{attribute addProperty BoxType "EK1100-0000-0018"}
{attribute addProperty Id "Beckhoff_ELXxxxxEK1122Beckhoff_ELXxxxxEK1122_CE175A58162A_0001_ELX1052_0000_0016ELX1052_F21EA95A506.25A_0002_ELX1054_0000_0016ELX1054_E012CCE111414.25A_0003_ELX1058_0000_0016ELX1058_D4A7C46F21026.25A_0004_ELX2002_0000_0016ELX2002_39EC201D334.125A_0005_ELX2008_0000_0016ELX2008_A854BE6D8110.125A_0006_ELX3152_0000_0016ELX3152_C6F348DD14618.25A_0007_ELX3152_0000_0017ELX3152_C6F348DD14618.25A_0008_ELX3152_0090_0016ELX3152_C6F348DD14618.25A_0009_ELX3152_0090_0017ELX3152_C6F348DD14618.25A_0010_ELX3158_0000_0016ELX3158_060F55FF33842.25A_0011_ELX3181_0000_0016ELX3181_644058BD16220.25A_0012_ELX3181_0000_0017ELX3181_644058BD16220.25A_0013_ELX3202_0000_0016ELX3202_4309805B14618.25A_0014_ELX3202_0090_0016ELX3202_4309805B14618.25A_0015_ELX3204_0000_0016ELX3204_B9E4353021026.25A_0016_ELX3204_0090_0016ELX3204_B9E4353021026.25A_0017_ELX3252_0000_0016ELX3252_CE5FC2FF14618.25A_0018_ELX3312_0000_0016ELX3312_92F3213114618.25A_0019_ELX3312_0090_0016ELX3312_92F3213114618.25A_0020_ELX3314_0000_0016ELX3314_A69716D721026.25A_0021_ELX3314_0090_0016ELX3314_A69716D721026.25A_0022_ELX3351_0000_0016ELX3351_9C5D626314618.25A_0023_ELX3351_0090_0016ELX3351_9C5D626314618.25A_0024_ELX4154_0000_0016ELX4154_9786CACB14518.125A_0025_ELX4181_0000_0016ELX4181_F21B729814518.125A_0026_ELX4181_0000_0017ELX4181_F21B729814518.125A_0027_ELX5151_0000_0016ELX5151_C54C90A514618.25A_0028_ELX5151_0090_0016ELX5151_C54C90A514618.25A_0030_ELX9410_0000_0016ELX9410_0EEAC8F2344.25A_0031_ELX9410_0000_0017ELX9410_0EEAC8F2344.25A_0032_ELX9410_0000_0018ELX9410_B5764C82344.25A_0033_ELX9560_0000_0016ELX9560_439807EB344.25A_0034_ELX9560_0000_0017ELX9560_439807EB344.25A_0035_ELX9560_0000_0018ELX9560_AB2C9EC5344.25"}
{attribute addProperty CRC "153078408"}
{attribute addProperty SizeInBites "4543"}
{attribute addProperty SizeInBytes "567.875"}
TYPE Beckhoff_ELXxxxx_091FCA88 EXTENDS EK1100_179A0949 :
STRUCT
	{attribute addProperty Name "Beckhoff_ELXxxxxEK1122"}
	Beckhoff_ELXxxxxEK1122 : Beckhoff_ELXxxxxEK1122_CE175A58;
	{attribute addProperty Name "A_0001_ELX1052_0000_0016"}
	A_0001_ELX1052_0000_0016 : ELX1052_F21EA95A;
	{attribute addProperty Name "A_0002_ELX1054_0000_0016"}
	A_0002_ELX1054_0000_0016 : ELX1054_E012CCE1;
	{attribute addProperty Name "A_0003_ELX1058_0000_0016"}
	A_0003_ELX1058_0000_0016 : ELX1058_D4A7C46F;
	{attribute addProperty Name "A_0004_ELX2002_0000_0016"}
	A_0004_ELX2002_0000_0016 : ELX2002_39EC201D;
	{attribute addProperty Name "A_0005_ELX2008_0000_0016"}
	A_0005_ELX2008_0000_0016 : ELX2008_A854BE6D;
	{attribute addProperty Name "A_0006_ELX3152_0000_0016"}
	A_0006_ELX3152_0000_0016 : ELX3152_C6F348DD;
	{attribute addProperty Name "A_0007_ELX3152_0000_0017"}
	A_0007_ELX3152_0000_0017 : ELX3152_C6F348DD;
	{attribute addProperty Name "A_0008_ELX3152_0090_0016"}
	A_0008_ELX3152_0090_0016 : ELX3152_C6F348DD;
	{attribute addProperty Name "A_0009_ELX3152_0090_0017"}
	A_0009_ELX3152_0090_0017 : ELX3152_C6F348DD;
	{attribute addProperty Name "A_0010_ELX3158_0000_0016"}
	A_0010_ELX3158_0000_0016 : ELX3158_060F55FF;
	{attribute addProperty Name "A_0011_ELX3181_0000_0016"}
	A_0011_ELX3181_0000_0016 : ELX3181_644058BD;
	{attribute addProperty Name "A_0012_ELX3181_0000_0017"}
	A_0012_ELX3181_0000_0017 : ELX3181_644058BD;
	{attribute addProperty Name "A_0013_ELX3202_0000_0016"}
	A_0013_ELX3202_0000_0016 : ELX3202_4309805B;
	{attribute addProperty Name "A_0014_ELX3202_0090_0016"}
	A_0014_ELX3202_0090_0016 : ELX3202_4309805B;
	{attribute addProperty Name "A_0015_ELX3204_0000_0016"}
	A_0015_ELX3204_0000_0016 : ELX3204_B9E43530;
	{attribute addProperty Name "A_0016_ELX3204_0090_0016"}
	A_0016_ELX3204_0090_0016 : ELX3204_B9E43530;
	{attribute addProperty Name "A_0017_ELX3252_0000_0016"}
	A_0017_ELX3252_0000_0016 : ELX3252_CE5FC2FF;
	{attribute addProperty Name "A_0018_ELX3312_0000_0016"}
	A_0018_ELX3312_0000_0016 : ELX3312_92F32131;
	{attribute addProperty Name "A_0019_ELX3312_0090_0016"}
	A_0019_ELX3312_0090_0016 : ELX3312_92F32131;
	{attribute addProperty Name "A_0020_ELX3314_0000_0016"}
	A_0020_ELX3314_0000_0016 : ELX3314_A69716D7;
	{attribute addProperty Name "A_0021_ELX3314_0090_0016"}
	A_0021_ELX3314_0090_0016 : ELX3314_A69716D7;
	{attribute addProperty Name "A_0022_ELX3351_0000_0016"}
	A_0022_ELX3351_0000_0016 : ELX3351_9C5D6263;
	{attribute addProperty Name "A_0023_ELX3351_0090_0016"}
	A_0023_ELX3351_0090_0016 : ELX3351_9C5D6263;
	{attribute addProperty Name "A_0024_ELX4154_0000_0016"}
	A_0024_ELX4154_0000_0016 : ELX4154_9786CACB;
	{attribute addProperty Name "A_0025_ELX4181_0000_0016"}
	A_0025_ELX4181_0000_0016 : ELX4181_F21B7298;
	{attribute addProperty Name "A_0026_ELX4181_0000_0017"}
	A_0026_ELX4181_0000_0017 : ELX4181_F21B7298;
	{attribute addProperty Name "A_0027_ELX5151_0000_0016"}
	A_0027_ELX5151_0000_0016 : ELX5151_C54C90A5;
	{attribute addProperty Name "A_0028_ELX5151_0090_0016"}
	A_0028_ELX5151_0090_0016 : ELX5151_C54C90A5;
	{attribute addProperty Name "A_0030_ELX9410_0000_0016"}
	A_0030_ELX9410_0000_0016 : ELX9410_0EEAC8F2;
	{attribute addProperty Name "A_0031_ELX9410_0000_0017"}
	A_0031_ELX9410_0000_0017 : ELX9410_0EEAC8F2;
	{attribute addProperty Name "A_0032_ELX9410_0000_0018"}
	A_0032_ELX9410_0000_0018 : ELX9410_B5764C82;
	{attribute addProperty Name "A_0033_ELX9560_0000_0016"}
	A_0033_ELX9560_0000_0016 : ELX9560_439807EB;
	{attribute addProperty Name "A_0034_ELX9560_0000_0017"}
	A_0034_ELX9560_0000_0017 : ELX9560_439807EB;
	{attribute addProperty Name "A_0035_ELX9560_0000_0018"}
	A_0035_ELX9560_0000_0018 : ELX9560_AB2C9EC5;
END_STRUCT
END_TYPE

(* stored: Version 1.2.0.0, ProductVersion 3.1.4024.9
   DUT Beckhoff_ELXxxxx_091FCA88: Id {9de28fc3-8a83-4aa2-847c-b9ccd2f4ac89} *)
